{attribute 'qualified_only'}
{attribute 'to_string'}
TYPE E_GROUP_CHECK :
(
  CHECK_NULL,
  CHECK_GROUP_REF_INVALID := 10,
  CHECK_AXIS_REF_INVALID,
  CHECK_CTRL_INVALID,
  CHECK_STATE_INVALID,
  CHECK_Mover_ITF_REF_INVALID,
  CHECK_XPU_INFO_REF_INVALID,


  CHECK_ERROR             :=  9000,
  CHECK_DONE              := 10000
)UINT;
END_TYPE

(* stored: Version 1.1.0.1, ProductVersion 3.1.4026.13
   DUT E_GROUP_CHECK: Id {042a55f2-2a33-4a17-836f-e4290f0c05e2} *)
